// SIMATIC S7-200 project (STEP 7-Micro/WIN), CPU 224 CN REL 02.01

ORGANIZATION_BLOCK 主程序:OB1
TITLE=程序注释
BEGIN
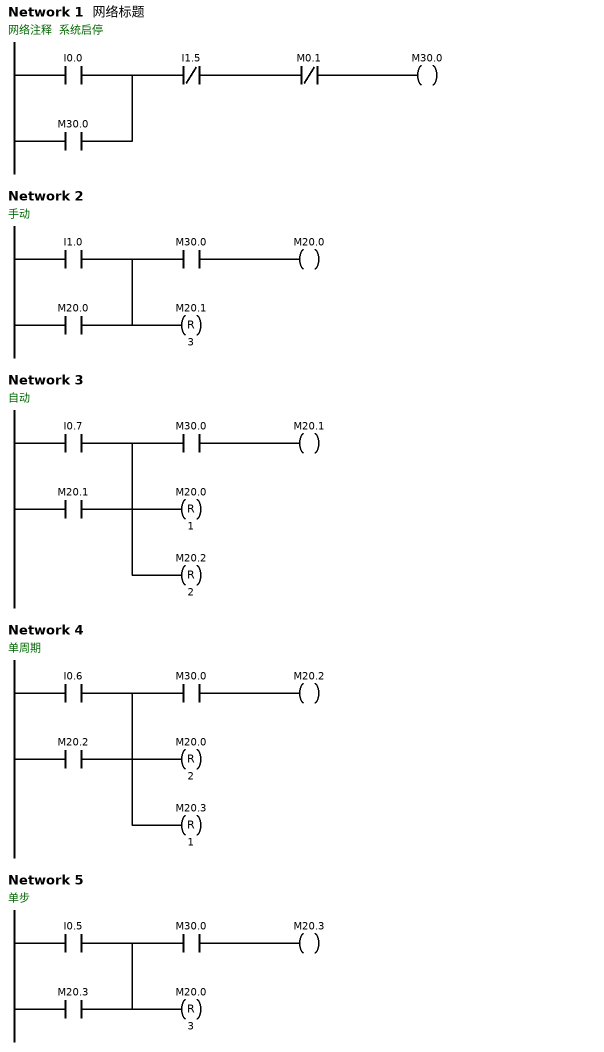
Network 1 // 网络标题
// 网络注释	系统启停
LD     I0.0
O      M30.0
AN     I1.5
AN     M0.1
=      M30.0
Network 2
// 手动	
LD     I1.0
O      M20.0
LPS
A      M30.0
=      M20.0
LPP
R      M20.1, 3
Network 3
// 自动
LD     I0.7
O      M20.1
LPS
A      M30.0
=      M20.1
LRD
R      M20.0, 1
LPP
R      M20.2, 2
Network 4
// 单周期
LD     I0.6
O      M20.2
LPS
A      M30.0
=      M20.2
LRD
R      M20.0, 2
LPP
R      M20.3, 1
Network 5
// 单步
LD     I0.5
O      M20.3
LPS
A      M30.0
=      M20.3
LPP
R      M20.0, 3
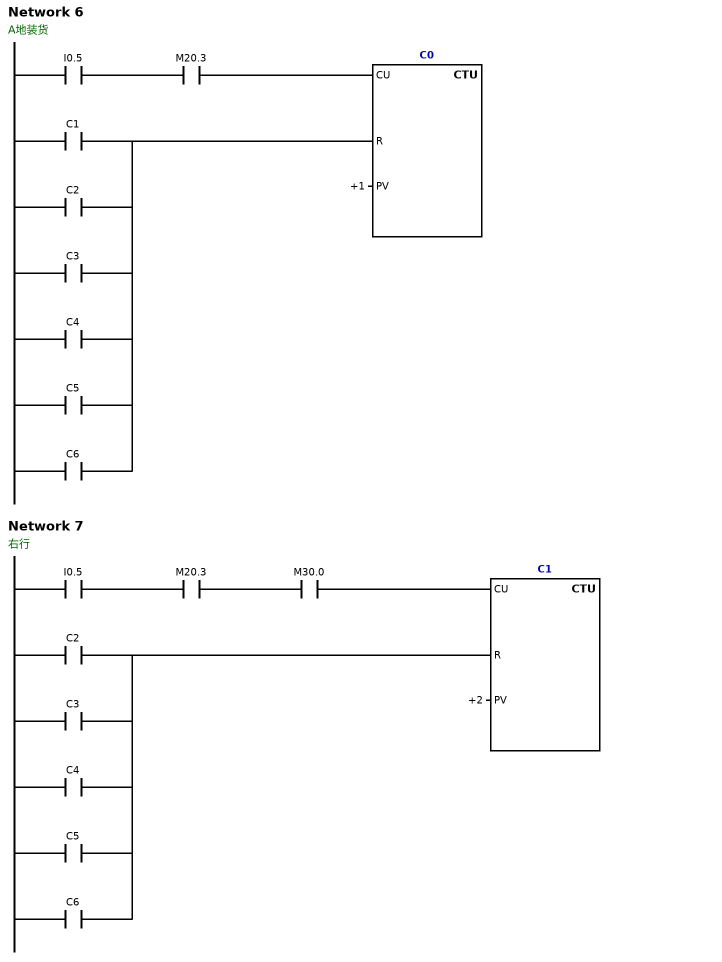
Network 6
// A地装货
LD     I0.5
A      M20.3
LD     C1
O      C2
O      C3
O      C4
O      C5
O      C6
CTU    C0, +1
Network 7
// 右行
LD     I0.5
A      M20.3
A      M30.0
LD     C2
O      C3
O      C4
O      C5
O      C6
CTU    C1, +2
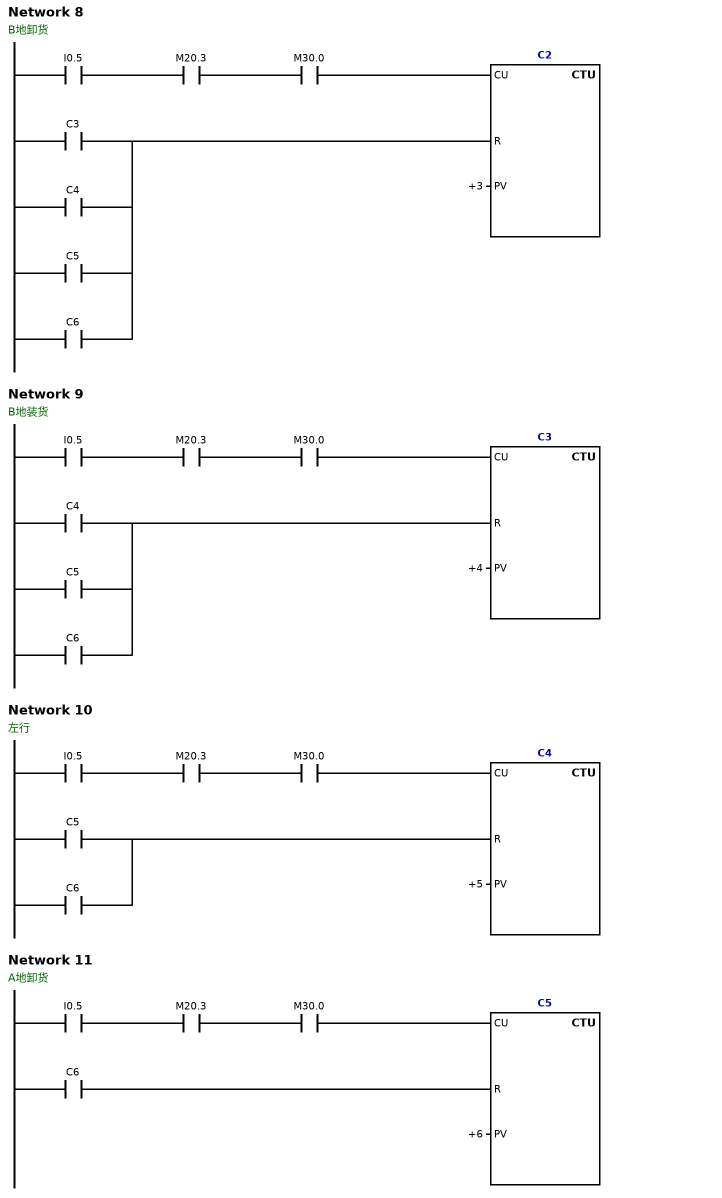
Network 8
// B地卸货
LD     I0.5
A      M20.3
A      M30.0
LD     C3
O      C4
O      C5
O      C6
CTU    C2, +3
Network 9
// B地装货
LD     I0.5
A      M20.3
A      M30.0
LD     C4
O      C5
O      C6
CTU    C3, +4
Network 10
// 左行
LD     I0.5
A      M20.3
A      M30.0
LD     C5
O      C6
CTU    C4, +5
Network 11
// A地卸货
LD     I0.5
A      M20.3
A      M30.0
LD     C6
CTU    C5, +6
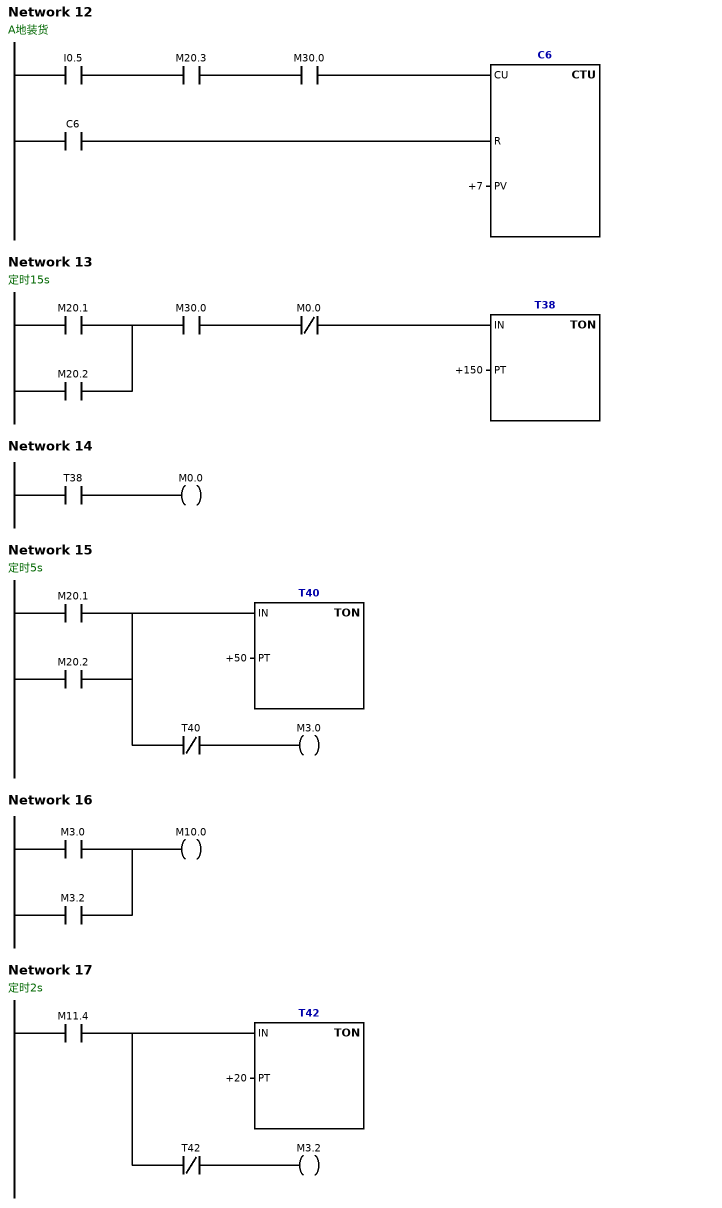
Network 12
// A地装货
LD     I0.5
A      M20.3
A      M30.0
LD     C6
CTU    C6, +7
Network 13
// 定时15s
LD     M20.1
O      M20.2
A      M30.0
AN     M0.0
TON    T38, +150
Network 14
LD     T38
=      M0.0
Network 15
// 定时5s
LD     M20.1
O      M20.2
TON    T40, +50
AN     T40
=      M3.0
Network 16
LD     M3.0
O      M3.2
=      M10.0
Network 17
// 定时2s
LD     M11.4
TON    T42, +20
AN     T42
=      M3.2
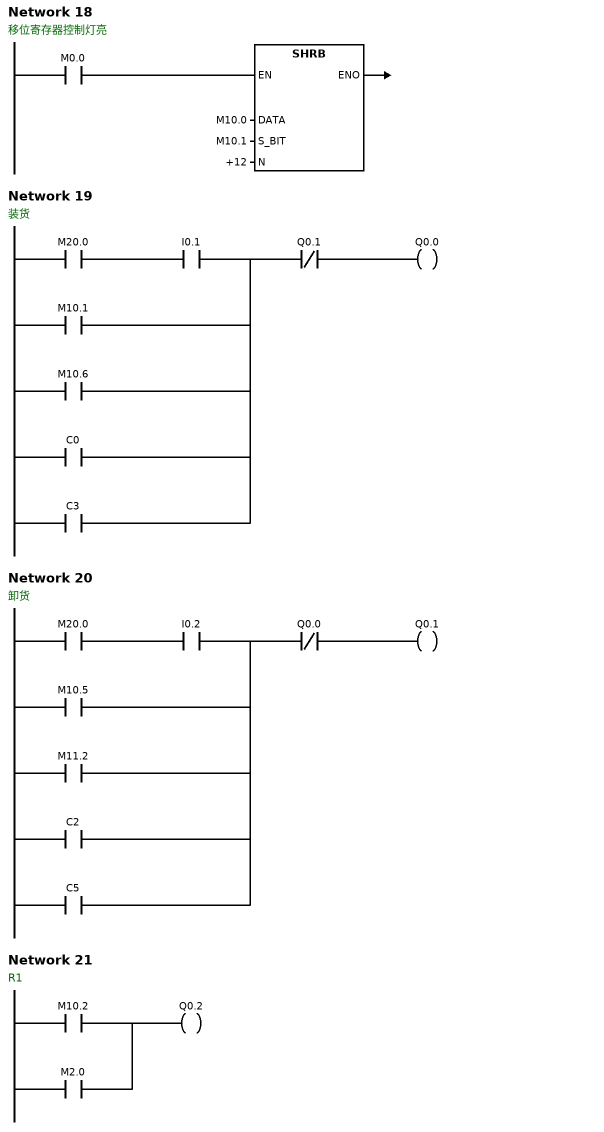
Network 18
// 移位寄存器控制灯亮
LD     M0.0
SHRB   M10.0, M10.1, +12
Network 19
// 装货
LD     M20.0
A      I0.1
O      M10.1
O      M10.6
O      C0
O      C3
AN     Q0.1
=      Q0.0
Network 20
// 卸货
LD     M20.0
A      I0.2
O      M10.5
O      M11.2
O      C2
O      C5
AN     Q0.0
=      Q0.1
Network 21
// R1
LD     M10.2
O      M2.0
=      Q0.2
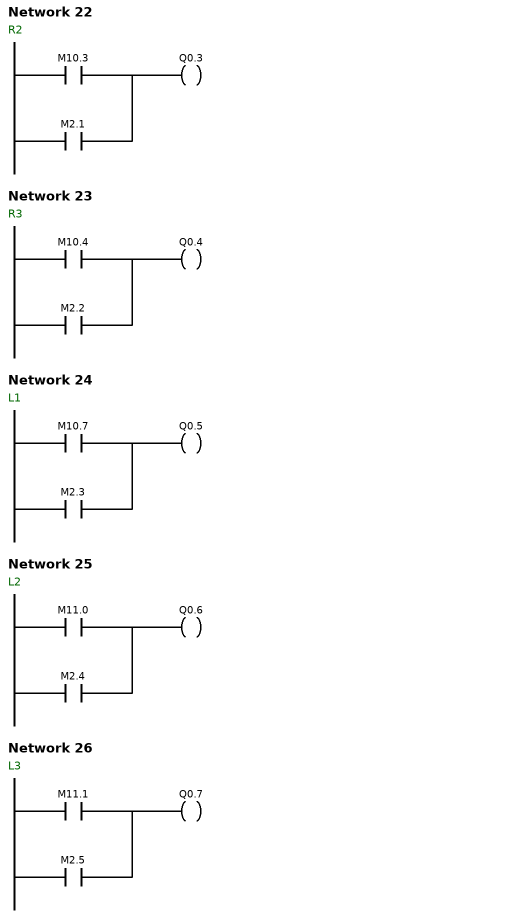
Network 22
// R2
LD     M10.3
O      M2.1
=      Q0.3
Network 23
// R3
LD     M10.4
O      M2.2
=      Q0.4
Network 24
// L1
LD     M10.7
O      M2.3
=      Q0.5
Network 25
// L2
LD     M11.0
O      M2.4
=      Q0.6
Network 26
// L3
LD     M11.1
O      M2.5
=      Q0.7
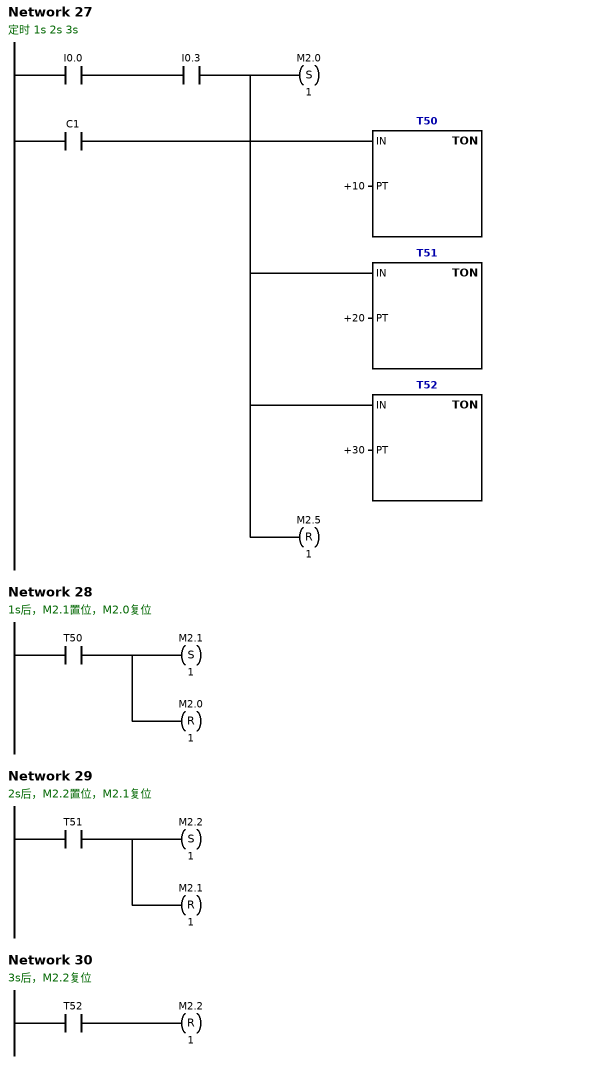
Network 27
// 定时 1s 2s 3s
LD     I0.0
A      I0.3
O      C1
S      M2.0, 1
TON    T50, +10
TON    T51, +20
TON    T52, +30
R      M2.5, 1
Network 28
// 1s后，M2.1置位，M2.0复位
LD     T50
S      M2.1, 1
R      M2.0, 1
Network 29
// 2s后，M2.2置位，M2.1复位
LD     T51
S      M2.2, 1
R      M2.1, 1
Network 30
// 3s后，M2.2复位
LD     T52
R      M2.2, 1
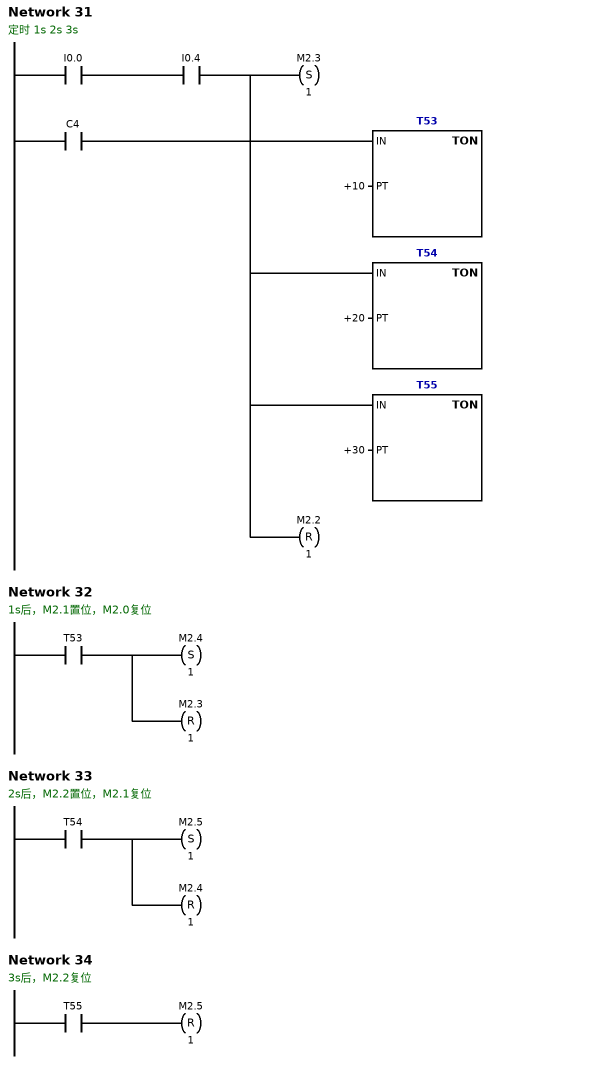
Network 31
// 定时 1s 2s 3s
LD     I0.0
A      I0.4
O      C4
S      M2.3, 1
TON    T53, +10
TON    T54, +20
TON    T55, +30
R      M2.2, 1
Network 32
// 1s后，M2.1置位，M2.0复位
LD     T53
S      M2.4, 1
R      M2.3, 1
Network 33
// 2s后，M2.2置位，M2.1复位
LD     T54
S      M2.5, 1
R      M2.4, 1
Network 34
// 3s后，M2.2复位
LD     T55
R      M2.5, 1
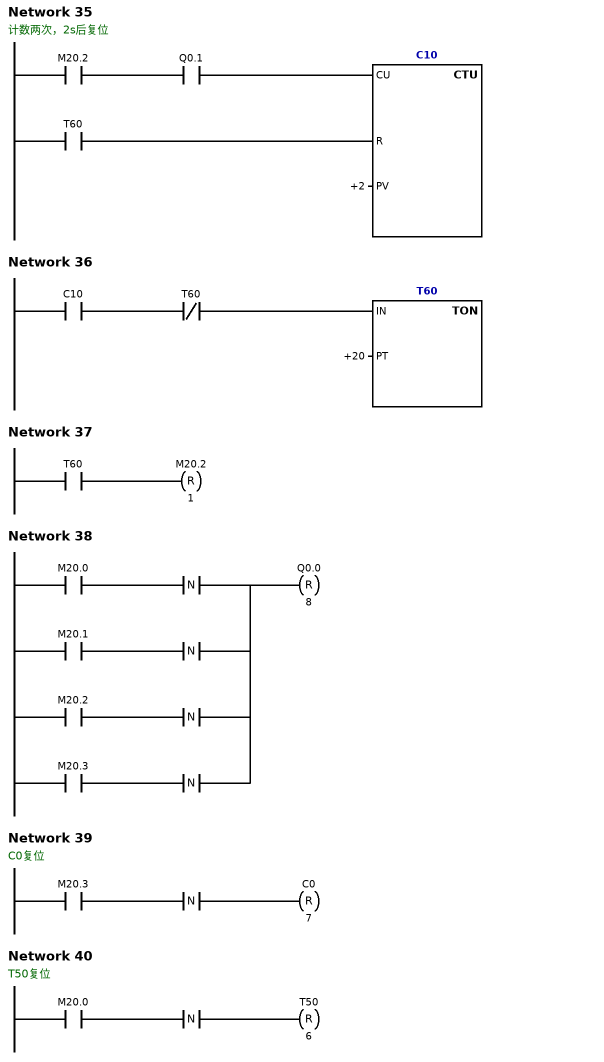
Network 35
// 计数两次，2s后复位
LD     M20.2
A      Q0.1
LD     T60
CTU    C10, +2
Network 36
LD     C10
AN     T60
TON    T60, +20
Network 37
LD     T60
R      M20.2, 1
Network 38
LD     M20.0
ED
LD     M20.1
ED
OLD
LD     M20.2
ED
OLD
LD     M20.3
ED
OLD
R      Q0.0, 8
Network 39
// C0复位
LD     M20.3
ED
R      C0, 7
Network 40
// T50复位
LD     M20.0
ED
R      T50, 6
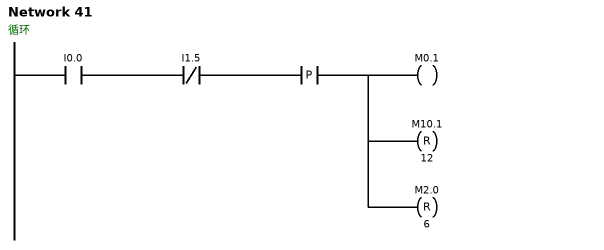
Network 41
// 循环
LD     I0.0
AN     I1.5
EU
=      M0.1
R      M10.1, 12
R      M2.0, 6
Network 43
// (network saved uncompiled; LAD cells follow)
// row 0: c0 ->
END_ORGANIZATION_BLOCK
